INTERFACE PUBLIC LoggingTargetAdapter EXTENDS __System.IQueryInterface

END_INTERFACE

(* stored: Version 1.1.0.1
   Itf LoggingTargetAdapter: Id {ac3659bf-3503-42a9-bb64-6b1d9ba4f3f5} *)
